FUNCTION_BLOCK FB_House

VAR
	   // Composition — Room created INSIDE House with its own constructor
    room    : FB_Room();  
    sOutput : STRING := '';
	sout4:STRING := '';
	
	{attribute 'hide'};
	x : INT :=55;
	
END_VAR

sout4 := 'checking';

METHOD showHouse
VAR_INPUT
END_VAR
sOutput := 'House contains a room';
END_METHOD

END_FUNCTION_BLOCK

(* stored: Version 1.1.0.1, ProductVersion 3.1.4024.16
   POU FB_House: Id {7c5f4edd-f1eb-4d8b-acb1-945195d2185d}, SpecialFunc None
   Method showHouse: Id {75c396d7-9ef7-41ca-8d69-8acc06e83a1a} *)
